Fanuc KAREL source: kt00204.KL

PROGRAM KT00204
%STACKSIZE=65535
%PRIORITY=65535
%NOLOCKGROUP
VAR
I1 : INTEGER
I2 : INTEGER
OUT : INTEGER
BEGIN
I1=2
I2=3
I1=2
I2=3
-- UNRESOLVED_PC line 12 opcodes [21 21 46 23] marker_code=64
END KT00204
